// TIA Portal V19 export
DATA_BLOCK "Ventil_Stati_DB"   // DB1095
// stored: AutoNumber false, InstanceOfName Ventil_Stati, InstanceOfType FB
"Ventil_Stati"
   // VAR RETAIN
   //    Param { ExternalAccessible := 'False'; ExternalVisible := 'False'; ExternalWritable := 'False'} : Struct
   //       "TO" : Time;
   //    END_STRUCT;
   //    Mld : Struct
   //       "TO_auf_CM01.QM18" : Bool;
   //       "TO_zu_CM01.QM18" : Bool;
   //       "SF_CM01.QM18" : Bool;
   //       "TO_auf_CM01.QM19" : Bool;
   //       "TO_zu_CM01.QM19" : Bool;
   //       "SF_CM01.QM19" : Bool;
   //       "TO_auf_CM01.QM20" : Bool;
   //       "TO_zu_CM01.QM20" : Bool;
   //       "SF_CM01.QM20" : Bool;
   //       "TO_auf_CM01.QM25" : Bool;
   //       "TO_zu_CM01.QM25" : Bool;
   //       "SF_CM01.QM25" : Bool;
   //       "TO_auf_CM01.QM26" : Bool;
   //       "TO_zu_CM01.QM26" : Bool;
   //       "SF_CM01.QM26" : Bool;
   //       "TO_auf_CM01.QM27" : Bool;
   //       "TO_zu_CM01.QM27" : Bool;
   //       "SF_CM01.QM27" : Bool;
   //       "TO_auf_CM02.QM55" : Bool;
   //       "TO_zu_CM02.QM55" : Bool;
   //       "SF_CM02.QM55" : Bool;
   //       "TO_auf_CM02.QM56" : Bool;
   //       "TO_zu_CM02.QM56" : Bool;
   //       "SF_CM02.QM56" : Bool;
   //       "TO_auf_CM02.QM57" : Bool;
   //       "TO_zu_CM02.QM57" : Bool;
   //       "SF_CM02.QM57" : Bool;
   //       "TO_auf_CM02.QM62" : Bool;
   //       "TO_zu_CM02.QM62" : Bool;
   //       "SF_CM02.QM62" : Bool;
   //       "TO_auf_CM02.QM63" : Bool;
   //       "TO_zu_CM02.QM63" : Bool;
   //       "SF_CM02.QM63" : Bool;
   //       "TO_auf_CM02.QM64" : Bool;
   //       "TO_zu_CM02.QM64" : Bool;
   //       "SF_CM02.QM64" : Bool;
   //       "TO_auf_HQ01.QM21" : Bool;
   //       "TO_zu_HQ01.QM21" : Bool;
   //       "SF_HQ01.QM21" : Bool;
   //       "TO_auf_HQ01.QM22" : Bool;
   //       "TO_zu_HQ01.QM22" : Bool;
   //       "SF_HQ01.QM22" : Bool;
   //       "TO_auf_HQ01.QM23" : Bool;
   //       "TO_zu_HQ01.QM23" : Bool;
   //       "SF_HQ01.QM23" : Bool;
   //       "TO_auf_HQ01.QM24" : Bool;
   //       "TO_zu_HQ01.QM24" : Bool;
   //       "SF_HQ01.QM24" : Bool;
   //       "TO_auf_HQ01.LV01" : Bool;
   //       "TO_zu_HQ01.LV01" : Bool;
   //       "SF_HQ01.LV01" : Bool;
   //       "TO_auf_HQ02.QM58" : Bool;
   //       "TO_zu_HQ02.QM58" : Bool;
   //       "SF_HQ02.QM58" : Bool;
   //       "TO_auf_HQ02.QM59" : Bool;
   //       "TO_zu_HQ02.QM59" : Bool;
   //       "SF_HQ02.QM59" : Bool;
   //       "TO_auf_HQ02.QM60" : Bool;
   //       "TO_zu_HQ02.QM60" : Bool;
   //       "SF_HQ02.QM60" : Bool;
   //       "TO_auf_HQ02.QM61" : Bool;
   //       "TO_zu_HQ02.QM61" : Bool;
   //       "SF_HQ02.QM61" : Bool;
   //       "TO_auf_HQ02.LV02" : Bool;
   //       "TO_zu_HQ02.LV02" : Bool;
   //       "SF_HQ02.LV02" : Bool;
   //       "TO_auf_CM03.QM33" : Bool;
   //       "TO_zu_CM03.QM33" : Bool;
   //       "SF_CM03.QM33" : Bool;
   //       "TO_auf_CM03.QM34" : Bool;
   //       "TO_zu_CM03.QM34" : Bool;
   //       "SF_CM03.QM34" : Bool;
   //       "TO_auf_CM04.QM72" : Bool;
   //       "TO_zu_CM04.QM72" : Bool;
   //       "SF_CM04.QM72" : Bool;
   //       "TO_auf_CM04.QM73" : Bool;
   //       "TO_zu_CM04.QM73" : Bool;
   //       "SF_CM04.QM73" : Bool;
   //       "TO_auf_CM05.QM61" : Bool;
   //       "TO_zu_CM05.QM61" : Bool;
   //       "SF_CM05.QM61" : Bool;
   //       "TO_auf_CM05.QM64" : Bool;
   //       "TO_zu_CM05.QM64" : Bool;
   //       "SF_CM05.QM64" : Bool;
   //       "TO_auf_GP01.QM14" : Bool;
   //       "TO_zu_GP01.QM14" : Bool;
   //       "SF_GP01.QM14" : Bool;
   //       "TO_auf_GP01.QM15" : Bool;
   //       "TO_zu_GP01.QM15" : Bool;
   //       "SF_GP01.QM15" : Bool;
   //       "TO_auf_GP01.QM16" : Bool;
   //       "TO_zu_GP01.QM16" : Bool;
   //       "SF_GP01.QM16" : Bool;
   //       "TO_auf_GP01.QM17" : Bool;
   //       "TO_zu_GP01.QM17" : Bool;
   //       "SF_GP01.QM17" : Bool;
   //       "TO_auf_GP01.QM18" : Bool;
   //       "TO_zu_GP01.QM18" : Bool;
   //       "SF_GP01.QM18" : Bool;
   //       "TO_auf_GP01.QM19" : Bool;
   //       "TO_zu_GP01.QM19" : Bool;
   //       "SF_GP01.QM19" : Bool;
   //       "TO_auf_GP01.QM20" : Bool;
   //       "TO_zu_GP01.QM20" : Bool;
   //       "SF_GP01.QM20" : Bool;
   //       "TO_auf_GP01.QM21" : Bool;
   //       "TO_zu_GP01.QM21" : Bool;
   //       "SF_GP01.QM21" : Bool;
   //       "TO_auf_GP01.QM22" : Bool;
   //       "TO_zu_GP01.QM22" : Bool;
   //       "SF_GP01.QM22" : Bool;
   //       "TO_auf_GP02.QM38" : Bool;
   //       "TO_zu_GP02.QM38" : Bool;
   //       "SF_GP02.QM38" : Bool;
   //       "TO_auf_GP02.QM39" : Bool;
   //       "TO_zu_GP02.QM39" : Bool;
   //       "SF_GP02.QM39" : Bool;
   //       "TO_auf_GP02.QM40" : Bool;
   //       "TO_zu_GP02.QM40" : Bool;
   //       "SF_GP02.QM40" : Bool;
   //       "TO_auf_GP02.QM41" : Bool;
   //       "TO_zu_GP02.QM41" : Bool;
   //       "SF_GP02.QM41" : Bool;
   //       "TO_auf_GP02.QM42" : Bool;
   //       "TO_zu_GP02.QM42" : Bool;
   //       "SF_GP02.QM42" : Bool;
   //       "TO_auf_GP02.QM43" : Bool;
   //       "TO_zu_GP02.QM43" : Bool;
   //       "SF_GP02.QM43" : Bool;
   //       "TO_auf_GP02.QM44" : Bool;
   //       "TO_zu_GP02.QM44" : Bool;
   //       "SF_GP02.QM44" : Bool;
   //       "TO_auf_GP02.QM45" : Bool;
   //       "TO_zu_GP02.QM45" : Bool;
   //       "SF_GP02.QM45" : Bool;
   //       "TO_auf_GP02.QM46" : Bool;
   //       "TO_zu_GP02.QM46" : Bool;
   //       "SF_GP02.QM46" : Bool;
   //    END_STRUCT;
   // END_VAR
   // VAR
   //    IEC_Timer { ExternalAccessible := 'False'; ExternalVisible := 'False'; ExternalWritable := 'False'} : Struct
   //       "TO_auf_CM01.QM18" { S7_SetPoint := 'True'} : TON_TIME;
   //       "TO_zu_CM01.QM18" { S7_SetPoint := 'True'} : TON_TIME;
   //       "TO_auf_CM01.QM19" { S7_SetPoint := 'True'} : TON_TIME;
   //       "TO_zu_CM01.QM19" { S7_SetPoint := 'True'} : TON_TIME;
   //       "TO_auf_CM01.QM20" { S7_SetPoint := 'True'} : TON_TIME;
   //       "TO_zu_CM01.QM20" { S7_SetPoint := 'True'} : TON_TIME;
   //       "TO_auf_CM01.QM25" { S7_SetPoint := 'True'} : TON_TIME;
   //       "TO_zu_CM01.QM25" { S7_SetPoint := 'True'} : TON_TIME;
   //       "TO_auf_CM01.QM26" { S7_SetPoint := 'True'} : TON_TIME;
   //       "TO_zu_CM01.QM26" { S7_SetPoint := 'True'} : TON_TIME;
   //       "TO_auf_CM01.QM27" { S7_SetPoint := 'True'} : TON_TIME;
   //       "TO_zu_CM01.QM27" { S7_SetPoint := 'True'} : TON_TIME;
   //       "TO_auf_CM02.QM55" { S7_SetPoint := 'True'} : TON_TIME;
   //       "TO_zu_CM02.QM55" { S7_SetPoint := 'True'} : TON_TIME;
   //       "TO_auf_CM02.QM56" { S7_SetPoint := 'True'} : TON_TIME;
   //       "TO_zu_CM02.QM56" { S7_SetPoint := 'True'} : TON_TIME;
   //       "TO_auf_CM02.QM57" { S7_SetPoint := 'True'} : TON_TIME;
   //       "TO_zu_CM02.QM57" { S7_SetPoint := 'True'} : TON_TIME;
   //       "TO_auf_CM02.QM62" { S7_SetPoint := 'True'} : TON_TIME;
   //       "TO_zu_CM02.QM62" { S7_SetPoint := 'True'} : TON_TIME;
   //       "TO_auf_CM02.QM63" { S7_SetPoint := 'True'} : TON_TIME;
   //       "TO_zu_CM02.QM63" { S7_SetPoint := 'True'} : TON_TIME;
   //       "TO_auf_CM02.QM64" { S7_SetPoint := 'True'} : TON_TIME;
   //       "TO_zu_CM02.QM64" { S7_SetPoint := 'True'} : TON_TIME;
   //       "TO_auf_HQ01.QM21" { S7_SetPoint := 'True'} : TON_TIME;
   //       "TO_zu_HQ01.QM21" { S7_SetPoint := 'True'} : TON_TIME;
   //       "TO_auf_HQ01.QM22" { S7_SetPoint := 'True'} : TON_TIME;
   //       "TO_zu_HQ01.QM22" { S7_SetPoint := 'True'} : TON_TIME;
   //       "TO_auf_HQ01.QM23" { S7_SetPoint := 'True'} : TON_TIME;
   //       "TO_zu_HQ01.QM23" { S7_SetPoint := 'True'} : TON_TIME;
   //       "TO_auf_HQ01.QM24" { S7_SetPoint := 'True'} : TON_TIME;
   //       "TO_zu_HQ01.QM24" { S7_SetPoint := 'True'} : TON_TIME;
   //       "TO_auf_HQ01.LV01" { S7_SetPoint := 'True'} : TON_TIME;
   //       "TO_zu_HQ01.LV01" { S7_SetPoint := 'True'} : TON_TIME;
   //       "TO_auf_HQ02.QM58" { S7_SetPoint := 'True'} : TON_TIME;
   //       "TO_zu_HQ02.QM58" { S7_SetPoint := 'True'} : TON_TIME;
   //       "TO_auf_HQ02.QM59" { S7_SetPoint := 'True'} : TON_TIME;
   //       "TO_zu_HQ02.QM59" { S7_SetPoint := 'True'} : TON_TIME;
   //       "TO_auf_HQ02.QM60" { S7_SetPoint := 'True'} : TON_TIME;
   //       "TO_zu_HQ02.QM60" { S7_SetPoint := 'True'} : TON_TIME;
   //       "TO_auf_HQ02.QM61" { S7_SetPoint := 'True'} : TON_TIME;
   //       "TO_zu_HQ02.QM61" { S7_SetPoint := 'True'} : TON_TIME;
   //       "TO_auf_HQ02.LV02" { S7_SetPoint := 'True'} : TON_TIME;
   //       "TO_zu_HQ02.LV02" { S7_SetPoint := 'True'} : TON_TIME;
   //       "TO_auf_CM03.QM33" { S7_SetPoint := 'True'} : TON_TIME;
   //       "TO_zu_CM03.QM33" { S7_SetPoint := 'True'} : TON_TIME;
   //       "TO_auf_CM03.QM34" { S7_SetPoint := 'True'} : TON_TIME;
   //       "TO_zu_CM03.QM34" { S7_SetPoint := 'True'} : TON_TIME;
   //       "TO_auf_CM04.QM72" { S7_SetPoint := 'True'} : TON_TIME;
   //       "TO_zu_CM04.QM72" { S7_SetPoint := 'True'} : TON_TIME;
   //       "TO_auf_CM04.QM73" { S7_SetPoint := 'True'} : TON_TIME;
   //       "TO_zu_CM04.QM73" { S7_SetPoint := 'True'} : TON_TIME;
   //       "TO_auf_CM05.QM61" { S7_SetPoint := 'True'} : TON_TIME;
   //       "TO_zu_CM05.QM61" { S7_SetPoint := 'True'} : TON_TIME;
   //       "TO_auf_CM05.QM64" { S7_SetPoint := 'True'} : TON_TIME;
   //       "TO_zu_CM05.QM64" { S7_SetPoint := 'True'} : TON_TIME;
   //       "TO_auf_GP01.QM14" { S7_SetPoint := 'True'} : TON_TIME;
   //       "TO_zu_GP01.QM14" { S7_SetPoint := 'True'} : TON_TIME;
   //       "TO_auf_GP01.QM15" { S7_SetPoint := 'True'} : TON_TIME;
   //       "TO_zu_GP01.QM15" { S7_SetPoint := 'True'} : TON_TIME;
   //       "TO_auf_GP01.QM16" { S7_SetPoint := 'True'} : TON_TIME;
   //       "TO_zu_GP01.QM16" { S7_SetPoint := 'True'} : TON_TIME;
   //       "TO_auf_GP01.QM17" { S7_SetPoint := 'True'} : TON_TIME;
   //       "TO_zu_GP01.QM17" { S7_SetPoint := 'True'} : TON_TIME;
   //       "TO_auf_GP01.QM18" { S7_SetPoint := 'True'} : TON_TIME;
   //       "TO_zu_GP01.QM18" { S7_SetPoint := 'True'} : TON_TIME;
   //       "TO_auf_GP01.QM19" { S7_SetPoint := 'True'} : TON_TIME;
   //       "TO_zu_GP01.QM19" { S7_SetPoint := 'True'} : TON_TIME;
   //       "TO_auf_GP01.QM20" { S7_SetPoint := 'True'} : TON_TIME;
   //       "TO_zu_GP01.QM20" { S7_SetPoint := 'True'} : TON_TIME;
   //       "TO_auf_GP01.QM21" { S7_SetPoint := 'True'} : TON_TIME;
   //       "TO_zu_GP01.QM21" { S7_SetPoint := 'True'} : TON_TIME;
   //       "TO_auf_GP01.QM22" { S7_SetPoint := 'True'} : TON_TIME;
   //       "TO_zu_GP01.QM22" { S7_SetPoint := 'True'} : TON_TIME;
   //       "TO_auf_GP02.QM38" { S7_SetPoint := 'True'} : TON_TIME;
   //       "TO_zu_GP02.QM38" { S7_SetPoint := 'True'} : TON_TIME;
   //       "TO_auf_GP02.QM39" { S7_SetPoint := 'True'} : TON_TIME;
   //       "TO_zu_GP02.QM39" { S7_SetPoint := 'True'} : TON_TIME;
   //       "TO_auf_GP02.QM40" { S7_SetPoint := 'True'} : TON_TIME;
   //       "TO_zu_GP02.QM40" { S7_SetPoint := 'True'} : TON_TIME;
   //       "TO_auf_GP02.QM41" { S7_SetPoint := 'True'} : TON_TIME;
   //       "TO_zu_GP02.QM41" { S7_SetPoint := 'True'} : TON_TIME;
   //       "TO_auf_GP02.QM42" { S7_SetPoint := 'True'} : TON_TIME;
   //       "TO_zu_GP02.QM42" { S7_SetPoint := 'True'} : TON_TIME;
   //       "TO_auf_GP02.QM43" { S7_SetPoint := 'True'} : TON_TIME;
   //       "TO_zu_GP02.QM43" { S7_SetPoint := 'True'} : TON_TIME;
   //       "TO_auf_GP02.QM44" { S7_SetPoint := 'True'} : TON_TIME;
   //       "TO_zu_GP02.QM44" { S7_SetPoint := 'True'} : TON_TIME;
   //       "TO_auf_GP02.QM45" { S7_SetPoint := 'True'} : TON_TIME;
   //       "TO_zu_GP02.QM45" { S7_SetPoint := 'True'} : TON_TIME;
   //       "TO_auf_GP02.QM46" { S7_SetPoint := 'True'} : TON_TIME;
   //       "TO_zu_GP02.QM46" { S7_SetPoint := 'True'} : TON_TIME;
   //    END_STRUCT;
   // END_VAR
BEGIN
END_DATA_BLOCK
